FUNCTION_BLOCK FB_StartingAlarm
VAR_INPUT
	Start: BOOL;
	Stop: BOOL;
	AlarmOn: TIME := T#500MS;
	AlarmOff: TIME := T#500MS;
	AlarmCount: UINT := 3;
END_VAR
VAR_OUTPUT
	Run: BOOL;
	Busy: BOOL;
	StartAlarm: BOOL;
END_VAR
VAR
	eState: (eInit, eIdle, eStarting, eRunning);
	eAlarmState: (eAlarmInit, eAlarmOn, eAlarmOff, eAlarmDone);
	rtrigStart: R_TRIG;
	rtrigStop: R_TRIG;
	tonAlarmOn: TON;
	tonAlarmOff: TON;
	nAlarmCount: UINT;
END_VAR

// Triggers
rtrigStop(CLK := Stop);

// Stop Interrrupt
IF rtrigStop.Q THEN
	eState := eInit;
END_IF

// State Machine
CASE eState OF
	eInit:
		Run := FALSE;
		Busy := FALSE;
		StartAlarm := FALSE;
		eAlarmState := eAlarmInit;	
		eState := eIdle;
		
	eIdle:
		IF Start THEN
			eState := eStarting;
		END_IF
		
	eStarting:
		Busy := TRUE;
		
		// Abort if Start not Held
		IF NOT Start THEN
			eState := eInit;
		END_IF
		
		// Alarm Sequence
		CASE eAlarmState OF
			eAlarmInit:
				tonAlarmOn.IN := FALSE;
				tonAlarmOn.PT := AlarmOn;
				tonAlarmOff.IN := FALSE;
				tonAlarmOff.PT := AlarmOff;
				nAlarmCount := 0;
				eAlarmState := eAlarmOn;
			eAlarmOn:
				tonAlarmOn.IN := TRUE;
				StartAlarm := TRUE;
				IF tonAlarmOn.Q THEN
					tonAlarmOn.IN := FALSE;
					eAlarmState := eAlarmOff;
				END_IF
			eAlarmOff:
				tonAlarmOff.IN := TRUE;
				StartAlarm := FALSE;
				IF tonAlarmOff.Q THEN
					tonAlarmOff.IN := FALSE;
					nAlarmCount := nAlarmCount + 1;
					IF nAlarmCount < AlarmCount THEN
						eAlarmState := eAlarmOn;
					ELSE
						eAlarmState := eAlarmDone;
					END_IF
				END_IF
				
			eAlarmDone:
				eState := eRunning;
		END_CASE
		
	eRunning:
		Busy := FALSE;
		Run := TRUE;	
END_CASE

// Call Function Blocks
tonAlarmOn();
tonAlarmOff();

END_FUNCTION_BLOCK

(* stored: Version 1.1.0.1, ProductVersion 3.1.4024.12
   POU FB_StartingAlarm: Id {81e684f9-9e22-43ae-a22b-886186db1292}, SpecialFunc None *)
